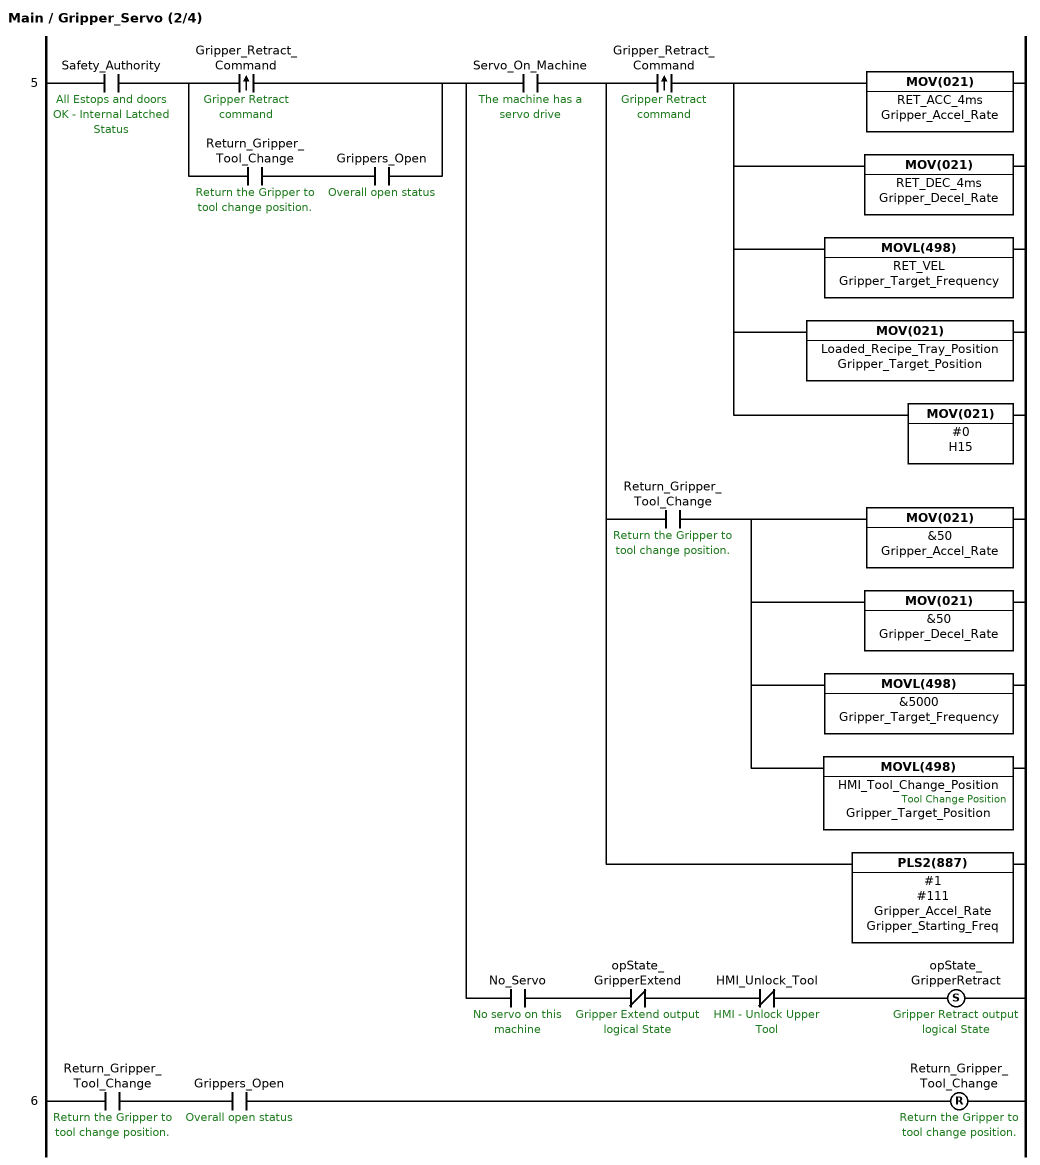
; [picture p96: Main / Gripper_Servo, rungs 5-6]
; rung 5
LD Safety_Authority  ; All Estops and doors OK - Internal Latched Status
@LD Gripper_Retract_Command  ; Gripper Retract command
LD Return_Gripper_Tool_Change  ; Return the Gripper to tool change position.
AND Grippers_Open  ; Overall open status
ORLD
ANDLD
OUT TR0
AND Servo_On_Machine  ; The machine has a servo drive
OUT TR1
@AND Gripper_Retract_Command  ; Gripper Retract command
MOV(021) RET_ACC_4ms Gripper_Accel_Rate
MOV(021) RET_DEC_4ms Gripper_Decel_Rate
MOVL(498) RET_VEL Gripper_Target_Frequency
MOV(021) Loaded_Recipe_Tray_Position Gripper_Target_Position
MOV(021) #0 H15
LD TR1
AND Return_Gripper_Tool_Change  ; Return the Gripper to tool change position.
MOV(021) &50 Gripper_Accel_Rate
MOV(021) &50 Gripper_Decel_Rate
MOVL(498) &5000 Gripper_Target_Frequency
MOVL(498) HMI_Tool_Change_Position Gripper_Target_Position  ; Tool Change Position
LD TR1
PLS2(887) #1 #111 Gripper_Accel_Rate Gripper_Starting_Freq
LD TR0
AND No_Servo  ; No servo on this machine
ANDNOT opState_GripperExtend  ; Gripper Extend output logical State
ANDNOT HMI_Unlock_Tool  ; HMI - Unlock Upper Tool
SET opState_GripperRetract  ; Gripper Retract output logical State
; rung 6
LD Return_Gripper_Tool_Change  ; Return the Gripper to tool change position.
AND Grippers_Open  ; Overall open status
RSET Return_Gripper_Tool_Change  ; Return the Gripper to tool change position.

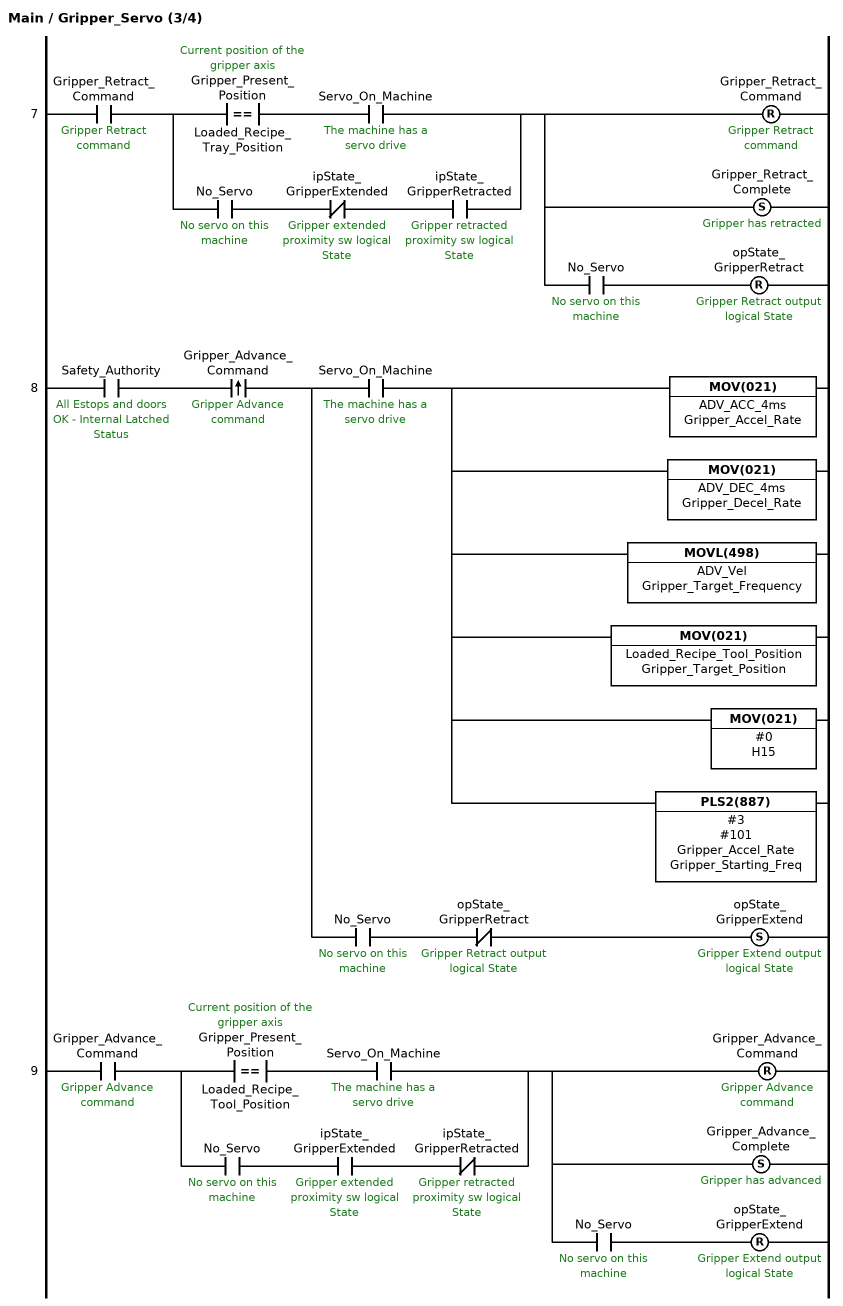
; rung 7
LD Gripper_Retract_Command  ; Gripper Retract command
LD=(300) Gripper_Present_Position Loaded_Recipe_Tray_Position  ; Current position of the gripper axis
AND Servo_On_Machine  ; The machine has a servo drive
LD No_Servo  ; No servo on this machine
ANDNOT ipState_GripperExtended  ; Gripper extended proximity sw logical State
AND ipState_GripperRetracted  ; Gripper retracted proximity sw logical State
ORLD
ANDLD
RSET Gripper_Retract_Command  ; Gripper Retract command
SET Gripper_Retract_Complete  ; Gripper has retracted
AND No_Servo  ; No servo on this machine
RSET opState_GripperRetract  ; Gripper Retract output logical State
; rung 8
LD Safety_Authority  ; All Estops and doors OK - Internal Latched Status
@AND Gripper_Advance_Command  ; Gripper Advance command
OUT TR0
AND Servo_On_Machine  ; The machine has a servo drive
MOV(021) ADV_ACC_4ms Gripper_Accel_Rate
MOV(021) ADV_DEC_4ms Gripper_Decel_Rate
MOVL(498) ADV_Vel Gripper_Target_Frequency
MOV(021) Loaded_Recipe_Tool_Position Gripper_Target_Position
MOV(021) #0 H15
PLS2(887) #3 #101 Gripper_Accel_Rate Gripper_Starting_Freq
LD TR0
AND No_Servo  ; No servo on this machine
ANDNOT opState_GripperRetract  ; Gripper Retract output logical State
SET opState_GripperExtend  ; Gripper Extend output logical State
; rung 9
LD Gripper_Advance_Command  ; Gripper Advance command
LD=(300) Gripper_Present_Position Loaded_Recipe_Tool_Position  ; Current position of the gripper axis
AND Servo_On_Machine  ; The machine has a servo drive
LD No_Servo  ; No servo on this machine
AND ipState_GripperExtended  ; Gripper extended proximity sw logical State
ANDNOT ipState_GripperRetracted  ; Gripper retracted proximity sw logical State
ORLD
ANDLD
RSET Gripper_Advance_Command  ; Gripper Advance command
SET Gripper_Advance_Complete  ; Gripper has advanced
AND No_Servo  ; No servo on this machine
RSET opState_GripperExtend  ; Gripper Extend output logical State

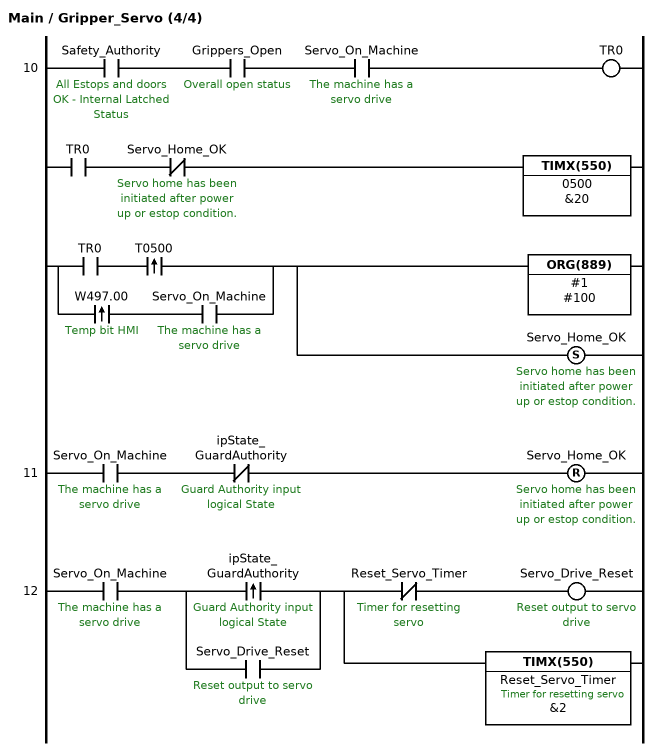
; rung 10
LD Safety_Authority  ; All Estops and doors OK - Internal Latched Status
AND Grippers_Open  ; Overall open status
AND Servo_On_Machine  ; The machine has a servo drive
OUT TR0
ANDNOT Servo_Home_OK  ; Servo home has been initiated after power up or estop condition.
TIMX(550) 0500 &20
LD TR0
@AND T0500
@LD W497.00  ; Temp bit HMI
AND Servo_On_Machine  ; The machine has a servo drive
ORLD
ORG(889) #1 #100
SET Servo_Home_OK  ; Servo home has been initiated after power up or estop condition.
; rung 11
LD Servo_On_Machine  ; The machine has a servo drive
ANDNOT ipState_GuardAuthority  ; Guard Authority input logical State
RSET Servo_Home_OK  ; Servo home has been initiated after power up or estop condition.
; rung 12
LD Servo_On_Machine  ; The machine has a servo drive
@LD ipState_GuardAuthority  ; Guard Authority input logical State
OR Servo_Drive_Reset  ; Reset output to servo drive
ANDLD
OUT TR0
ANDNOT Reset_Servo_Timer  ; Timer for resetting servo
OUT Servo_Drive_Reset  ; Reset output to servo drive
LD TR0
TIMX(550) Reset_Servo_Timer &2  ; Timer for resetting servo

### Section Temp_Control_and_Analog

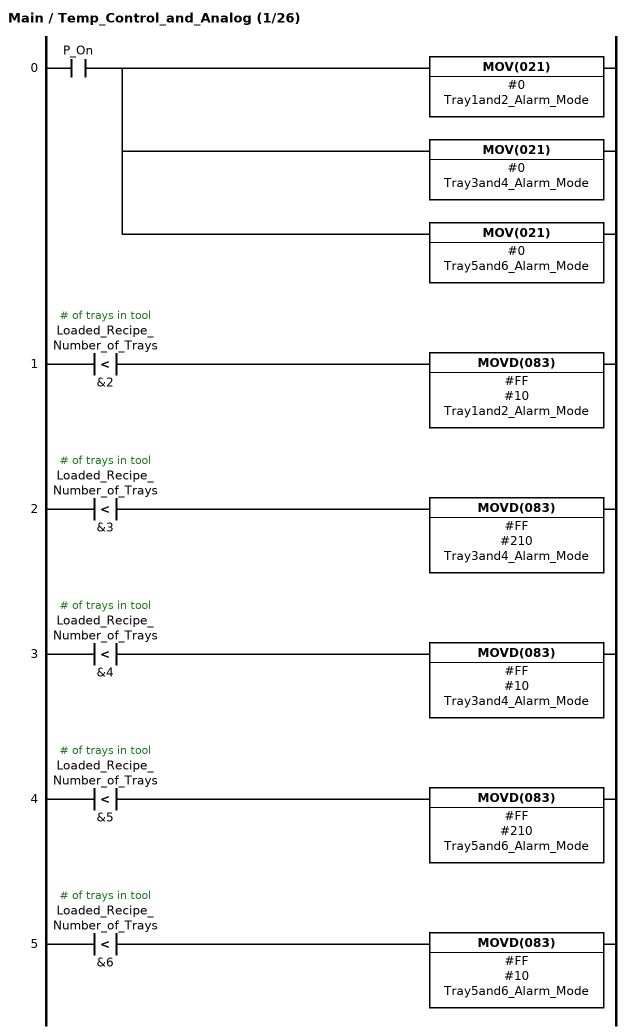
; rung 0
LD P_On
MOV(021) #0 Tray1and2_Alarm_Mode
MOV(021) #0 Tray3and4_Alarm_Mode
MOV(021) #0 Tray5and6_Alarm_Mode
; rung 1
LD<(310) Loaded_Recipe_Number_of_Trays &2  ; # of trays in tool
MOVD(083) #FF #10 Tray1and2_Alarm_Mode
; rung 2
LD<(310) Loaded_Recipe_Number_of_Trays &3  ; # of trays in tool
MOVD(083) #FF #210 Tray3and4_Alarm_Mode
; rung 3
LD<(310) Loaded_Recipe_Number_of_Trays &4  ; # of trays in tool
MOVD(083) #FF #10 Tray3and4_Alarm_Mode
; rung 4
LD<(310) Loaded_Recipe_Number_of_Trays &5  ; # of trays in tool
MOVD(083) #FF #210 Tray5and6_Alarm_Mode
; rung 5
LD<(310) Loaded_Recipe_Number_of_Trays &6  ; # of trays in tool
MOVD(083) #FF #10 Tray5and6_Alarm_Mode

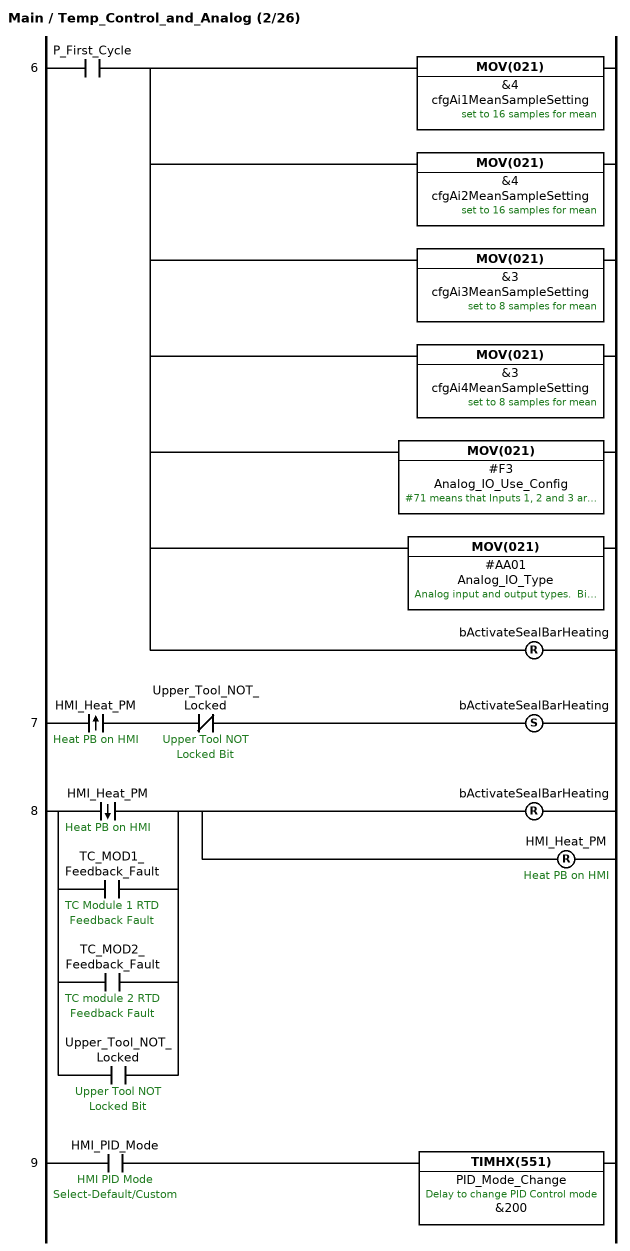
; rung 6
LD P_First_Cycle
MOV(021) &4 cfgAi1MeanSampleSetting  ; set to 16 samples for mean
MOV(021) &4 cfgAi2MeanSampleSetting  ; set to 16 samples for mean
MOV(021) &3 cfgAi3MeanSampleSetting  ; set to 8 samples for mean
MOV(021) &3 cfgAi4MeanSampleSetting  ; set to 8 samples for mean
MOV(021) #F3 Analog_IO_Use_Config  ; #71 means that Inputs 1, 2 and 3 are used (bits 4, 5 and 6 on makes up 7 HEX) and output 1 is used (bit 0 on makes up 1 HEX).
MOV(021) #AA01 Analog_IO_Type  ; Analog input and output types.  Bit pattern of 1010101000000001 (#AA01) means all inputs are 4-20 mA and the output are 0 - 10VDC).
RSET bActivateSealBarHeating
; rung 7
@LD HMI_Heat_PM  ; Heat PB on HMI
ANDNOT Upper_Tool_NOT_Locked  ; Upper Tool NOT Locked Bit
SET bActivateSealBarHeating
; rung 8
%LD HMI_Heat_PM  ; Heat PB on HMI
OR TC_MOD1_Feedback_Fault  ; TC Module 1 RTD Feedback Fault
OR TC_MOD2_Feedback_Fault  ; TC module 2 RTD Feedback Fault
OR Upper_Tool_NOT_Locked  ; Upper Tool NOT Locked Bit
RSET bActivateSealBarHeating
RSET HMI_Heat_PM  ; Heat PB on HMI
; rung 9
LD HMI_PID_Mode  ; HMI PID Mode Select-Default/Custom
TIMHX(551) PID_Mode_Change &200  ; Delay to change PID Control mode

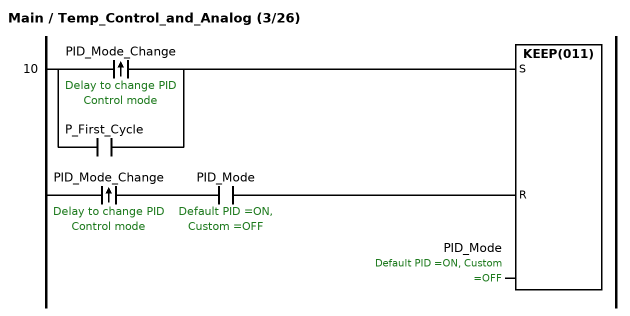
; rung 10
@LD PID_Mode_Change  ; Delay to change PID Control mode
OR P_First_Cycle
@LD PID_Mode_Change  ; Delay to change PID Control mode
AND PID_Mode  ; Default PID =ON, Custom =OFF
KEEP(011) PID_Mode  ; Default PID =ON, Custom =OFF

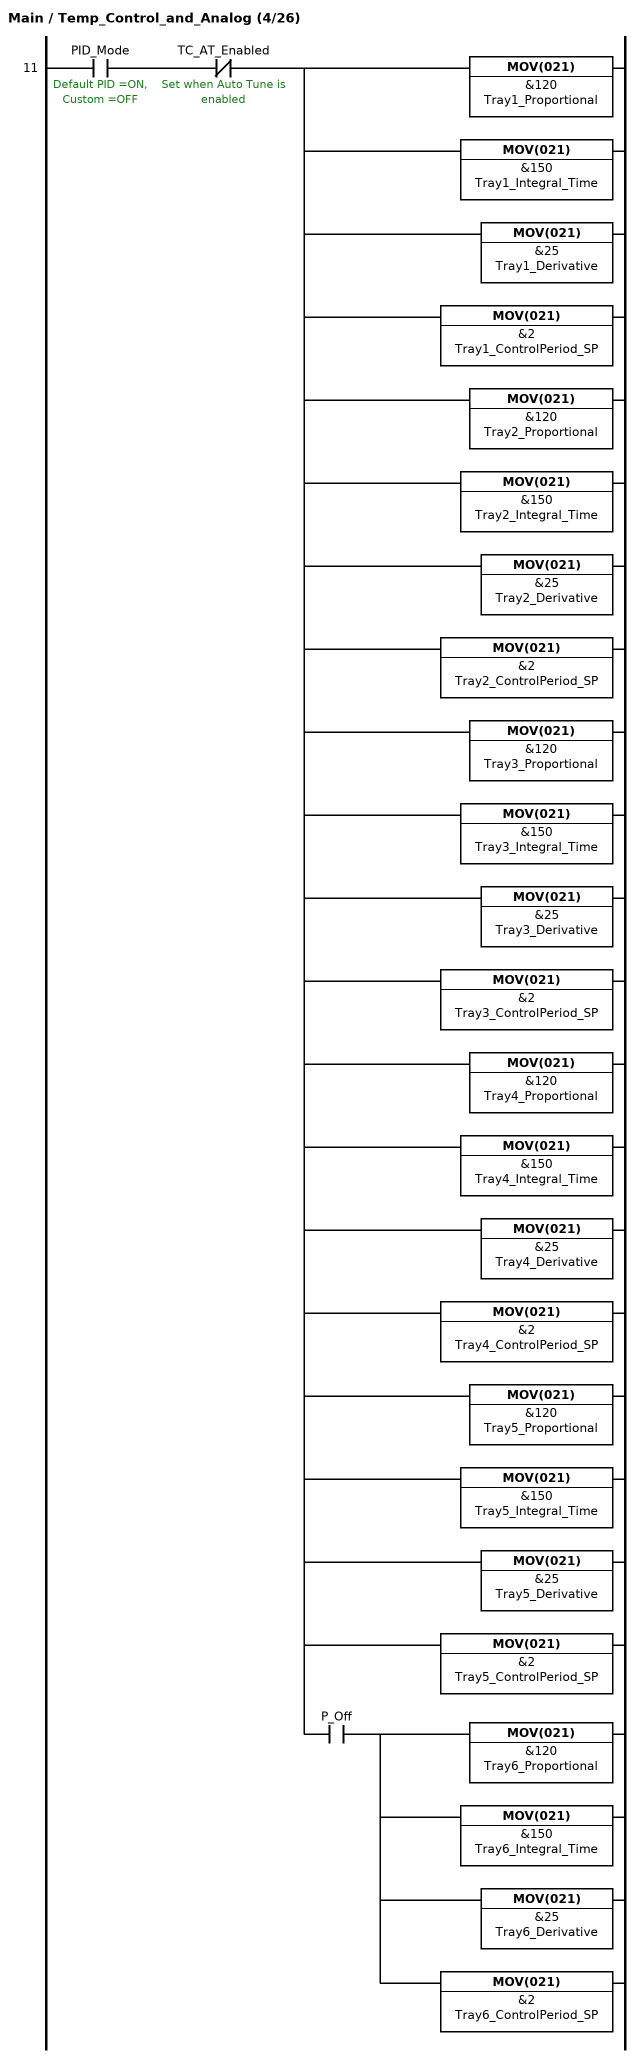
; rung 11
LD PID_Mode  ; Default PID =ON, Custom =OFF
ANDNOT TC_AT_Enabled  ; Set when Auto Tune is enabled
MOV(021) &120 Tray1_Proportional
MOV(021) &150 Tray1_Integral_Time
MOV(021) &25 Tray1_Derivative
MOV(021) &2 Tray1_ControlPeriod_SP
MOV(021) &120 Tray2_Proportional
MOV(021) &150 Tray2_Integral_Time
MOV(021) &25 Tray2_Derivative
MOV(021) &2 Tray2_ControlPeriod_SP
MOV(021) &120 Tray3_Proportional
MOV(021) &150 Tray3_Integral_Time
MOV(021) &25 Tray3_Derivative
MOV(021) &2 Tray3_ControlPeriod_SP
MOV(021) &120 Tray4_Proportional
MOV(021) &150 Tray4_Integral_Time
MOV(021) &25 Tray4_Derivative
MOV(021) &2 Tray4_ControlPeriod_SP
MOV(021) &120 Tray5_Proportional
MOV(021) &150 Tray5_Integral_Time
MOV(021) &25 Tray5_Derivative
MOV(021) &2 Tray5_ControlPeriod_SP
AND P_Off
MOV(021) &120 Tray6_Proportional
MOV(021) &150 Tray6_Integral_Time
MOV(021) &25 Tray6_Derivative
MOV(021) &2 Tray6_ControlPeriod_SP

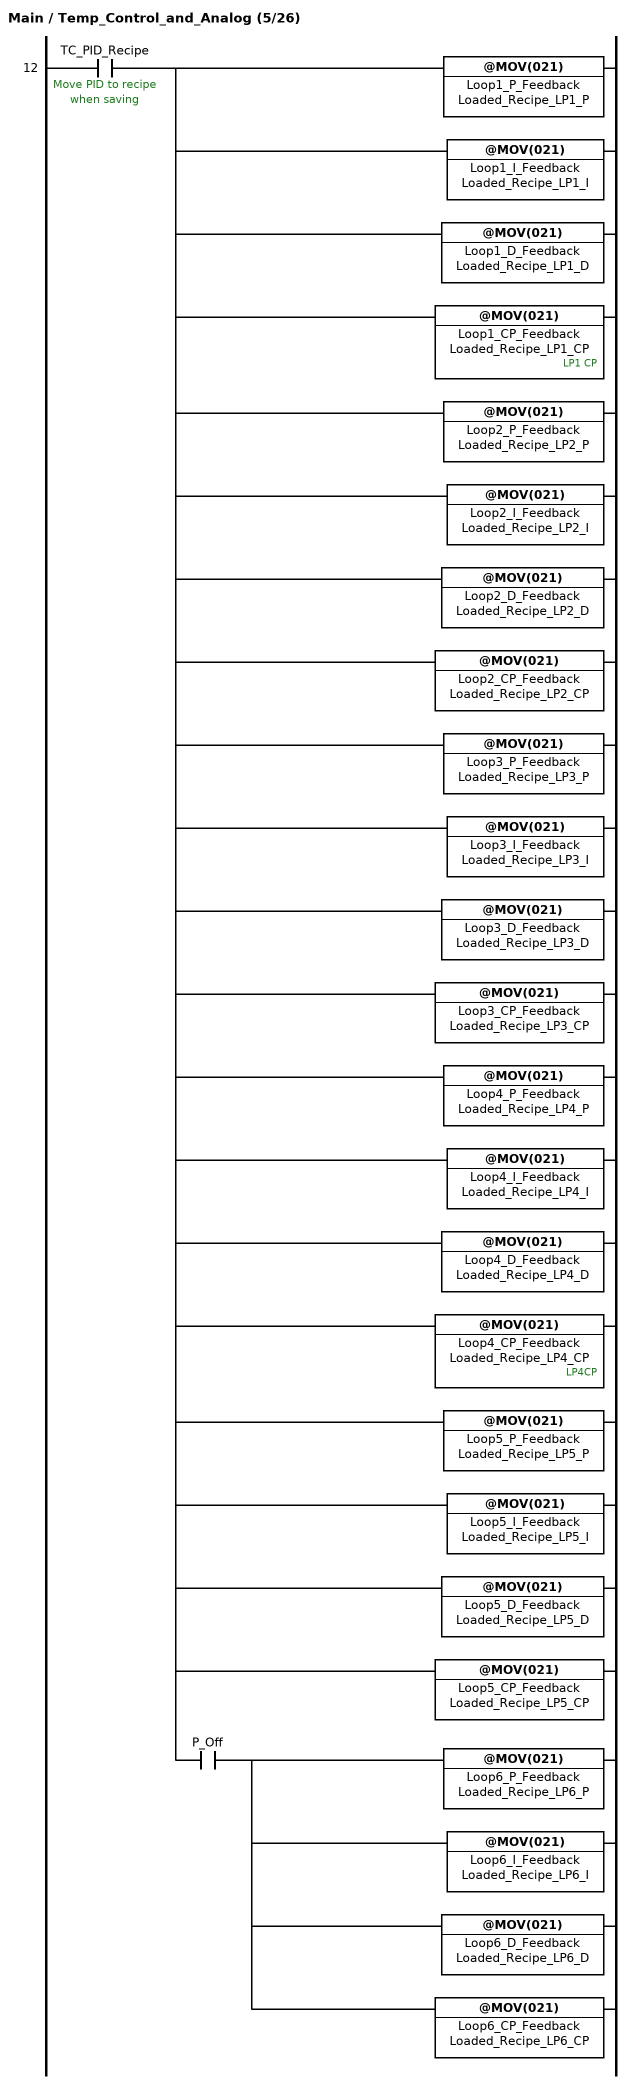
; rung 12
LD TC_PID_Recipe  ; Move PID to recipe when saving
@MOV(021) Loop1_P_Feedback Loaded_Recipe_LP1_P
@MOV(021) Loop1_I_Feedback Loaded_Recipe_LP1_I
@MOV(021) Loop1_D_Feedback Loaded_Recipe_LP1_D
@MOV(021) Loop1_CP_Feedback Loaded_Recipe_LP1_CP  ; LP1 CP
@MOV(021) Loop2_P_Feedback Loaded_Recipe_LP2_P
@MOV(021) Loop2_I_Feedback Loaded_Recipe_LP2_I
@MOV(021) Loop2_D_Feedback Loaded_Recipe_LP2_D
@MOV(021) Loop2_CP_Feedback Loaded_Recipe_LP2_CP
@MOV(021) Loop3_P_Feedback Loaded_Recipe_LP3_P
@MOV(021) Loop3_I_Feedback Loaded_Recipe_LP3_I
@MOV(021) Loop3_D_Feedback Loaded_Recipe_LP3_D
@MOV(021) Loop3_CP_Feedback Loaded_Recipe_LP3_CP
@MOV(021) Loop4_P_Feedback Loaded_Recipe_LP4_P
@MOV(021) Loop4_I_Feedback Loaded_Recipe_LP4_I
@MOV(021) Loop4_D_Feedback Loaded_Recipe_LP4_D
@MOV(021) Loop4_CP_Feedback Loaded_Recipe_LP4_CP  ; LP4CP
@MOV(021) Loop5_P_Feedback Loaded_Recipe_LP5_P
@MOV(021) Loop5_I_Feedback Loaded_Recipe_LP5_I
@MOV(021) Loop5_D_Feedback Loaded_Recipe_LP5_D
@MOV(021) Loop5_CP_Feedback Loaded_Recipe_LP5_CP
AND P_Off
@MOV(021) Loop6_P_Feedback Loaded_Recipe_LP6_P
@MOV(021) Loop6_I_Feedback Loaded_Recipe_LP6_I
@MOV(021) Loop6_D_Feedback Loaded_Recipe_LP6_D
@MOV(021) Loop6_CP_Feedback Loaded_Recipe_LP6_CP

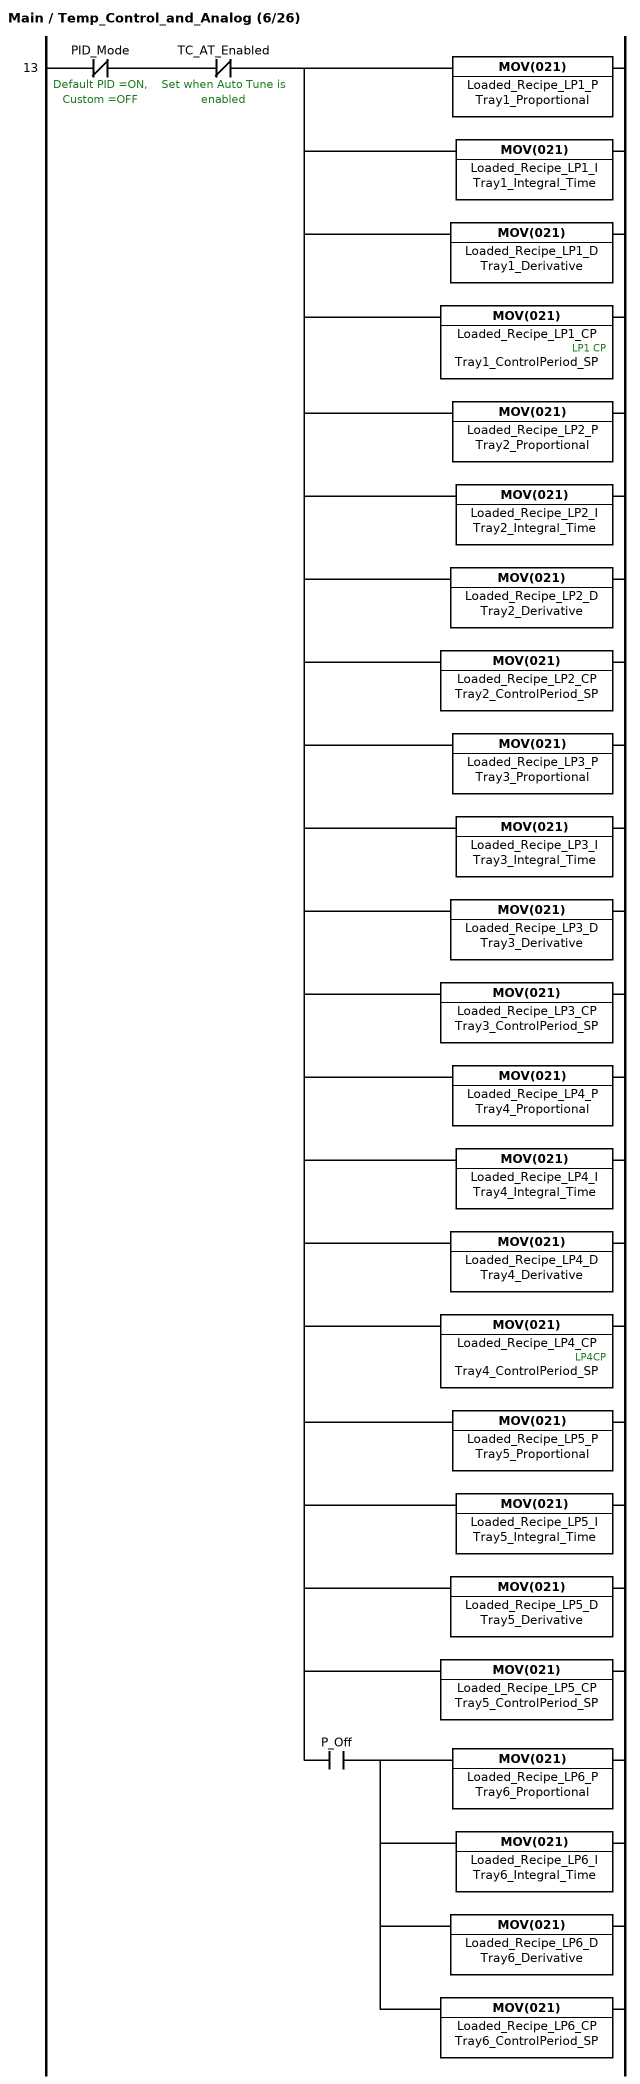
; rung 13
LDNOT PID_Mode  ; Default PID =ON, Custom =OFF
ANDNOT TC_AT_Enabled  ; Set when Auto Tune is enabled
MOV(021) Loaded_Recipe_LP1_P Tray1_Proportional
MOV(021) Loaded_Recipe_LP1_I Tray1_Integral_Time
MOV(021) Loaded_Recipe_LP1_D Tray1_Derivative
MOV(021) Loaded_Recipe_LP1_CP Tray1_ControlPeriod_SP  ; LP1 CP
MOV(021) Loaded_Recipe_LP2_P Tray2_Proportional
MOV(021) Loaded_Recipe_LP2_I Tray2_Integral_Time
MOV(021) Loaded_Recipe_LP2_D Tray2_Derivative
MOV(021) Loaded_Recipe_LP2_CP Tray2_ControlPeriod_SP
MOV(021) Loaded_Recipe_LP3_P Tray3_Proportional
MOV(021) Loaded_Recipe_LP3_I Tray3_Integral_Time
MOV(021) Loaded_Recipe_LP3_D Tray3_Derivative
MOV(021) Loaded_Recipe_LP3_CP Tray3_ControlPeriod_SP
MOV(021) Loaded_Recipe_LP4_P Tray4_Proportional
MOV(021) Loaded_Recipe_LP4_I Tray4_Integral_Time
MOV(021) Loaded_Recipe_LP4_D Tray4_Derivative
MOV(021) Loaded_Recipe_LP4_CP Tray4_ControlPeriod_SP  ; LP4CP
MOV(021) Loaded_Recipe_LP5_P Tray5_Proportional
MOV(021) Loaded_Recipe_LP5_I Tray5_Integral_Time
MOV(021) Loaded_Recipe_LP5_D Tray5_Derivative
MOV(021) Loaded_Recipe_LP5_CP Tray5_ControlPeriod_SP
AND P_Off
MOV(021) Loaded_Recipe_LP6_P Tray6_Proportional
MOV(021) Loaded_Recipe_LP6_I Tray6_Integral_Time
MOV(021) Loaded_Recipe_LP6_D Tray6_Derivative
MOV(021) Loaded_Recipe_LP6_CP Tray6_ControlPeriod_SP

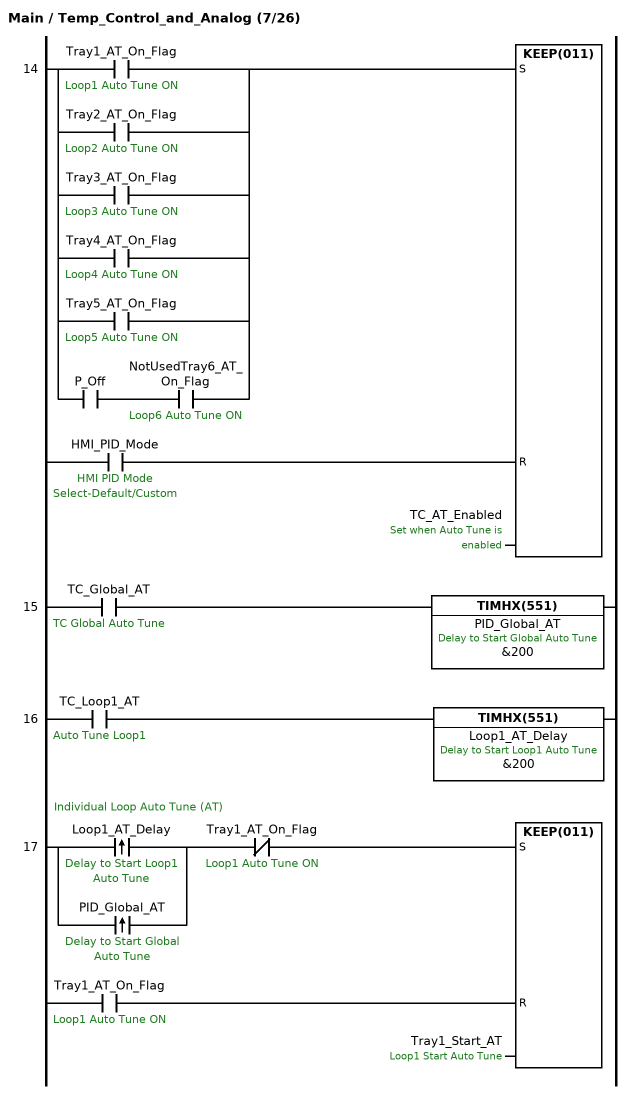
; rung 14
LD Tray1_AT_On_Flag  ; Loop1 Auto Tune ON
OR Tray2_AT_On_Flag  ; Loop2 Auto Tune ON
OR Tray3_AT_On_Flag  ; Loop3 Auto Tune ON
OR Tray4_AT_On_Flag  ; Loop4 Auto Tune ON
OR Tray5_AT_On_Flag  ; Loop5 Auto Tune ON
LD P_Off
AND NotUsedTray6_AT_On_Flag  ; Loop6 Auto Tune ON
ORLD
LD HMI_PID_Mode  ; HMI PID Mode Select-Default/Custom
KEEP(011) TC_AT_Enabled  ; Set when Auto Tune is enabled
; rung 15
LD TC_Global_AT  ; TC Global Auto Tune
TIMHX(551) PID_Global_AT &200  ; Delay to Start Global Auto Tune
; rung 16
LD TC_Loop1_AT  ; Auto Tune Loop1
TIMHX(551) Loop1_AT_Delay &200  ; Delay to Start Loop1 Auto Tune
; rung 17: Individual Loop Auto Tune (AT)
@LD Loop1_AT_Delay  ; Delay to Start Loop1 Auto Tune
@OR PID_Global_AT  ; Delay to Start Global Auto Tune
ANDNOT Tray1_AT_On_Flag  ; Loop1 Auto Tune ON
LD Tray1_AT_On_Flag  ; Loop1 Auto Tune ON
KEEP(011) Tray1_Start_AT  ; Loop1 Start Auto Tune

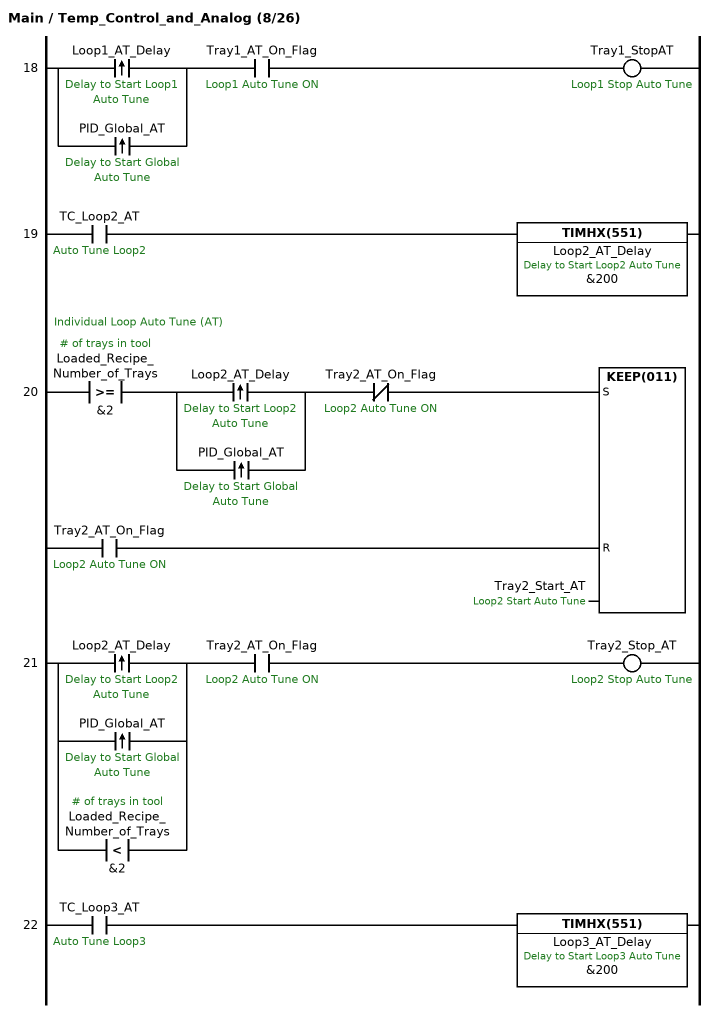
; rung 18
@LD Loop1_AT_Delay  ; Delay to Start Loop1 Auto Tune
@OR PID_Global_AT  ; Delay to Start Global Auto Tune
AND Tray1_AT_On_Flag  ; Loop1 Auto Tune ON
OUT Tray1_StopAT  ; Loop1 Stop Auto Tune
; rung 19
LD TC_Loop2_AT  ; Auto Tune Loop2
TIMHX(551) Loop2_AT_Delay &200  ; Delay to Start Loop2 Auto Tune
; rung 20: Individual Loop Auto Tune (AT)
LD>=(325) Loaded_Recipe_Number_of_Trays &2  ; # of trays in tool
@LD Loop2_AT_Delay  ; Delay to Start Loop2 Auto Tune
@OR PID_Global_AT  ; Delay to Start Global Auto Tune
ANDLD
ANDNOT Tray2_AT_On_Flag  ; Loop2 Auto Tune ON
LD Tray2_AT_On_Flag  ; Loop2 Auto Tune ON
KEEP(011) Tray2_Start_AT  ; Loop2 Start Auto Tune
; rung 21
@LD Loop2_AT_Delay  ; Delay to Start Loop2 Auto Tune
@OR PID_Global_AT  ; Delay to Start Global Auto Tune
OR<(310) Loaded_Recipe_Number_of_Trays &2  ; # of trays in tool
AND Tray2_AT_On_Flag  ; Loop2 Auto Tune ON
OUT Tray2_Stop_AT  ; Loop2 Stop Auto Tune
; rung 22
LD TC_Loop3_AT  ; Auto Tune Loop3
TIMHX(551) Loop3_AT_Delay &200  ; Delay to Start Loop3 Auto Tune

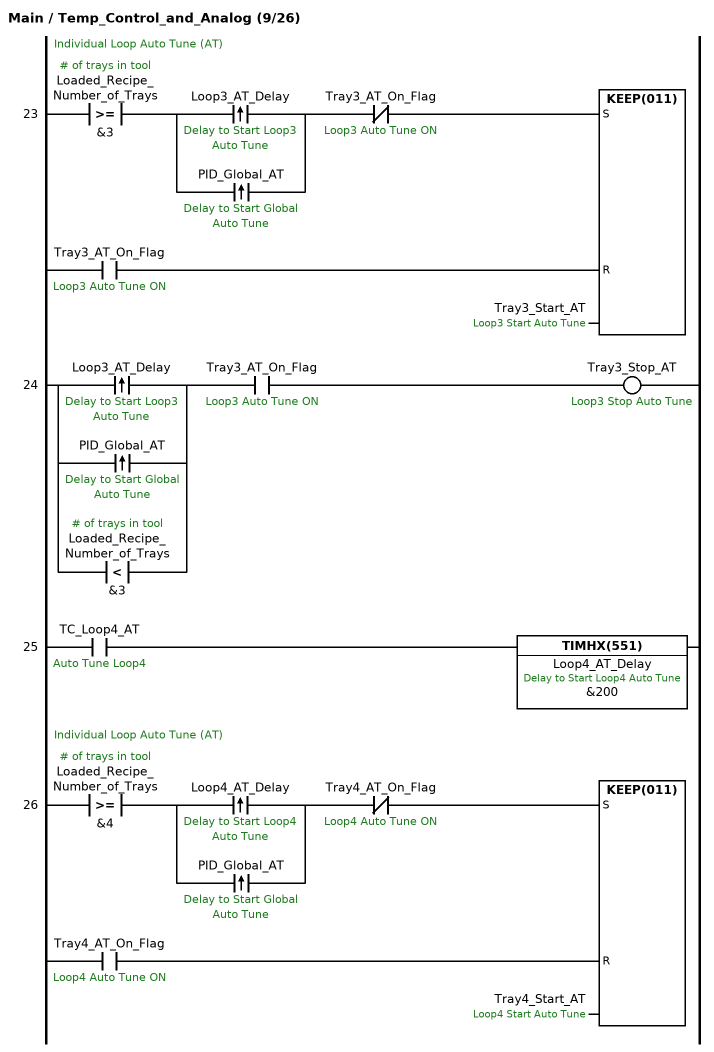
; rung 23: Individual Loop Auto Tune (AT)
LD>=(325) Loaded_Recipe_Number_of_Trays &3  ; # of trays in tool
@LD Loop3_AT_Delay  ; Delay to Start Loop3 Auto Tune
@OR PID_Global_AT  ; Delay to Start Global Auto Tune
ANDLD
ANDNOT Tray3_AT_On_Flag  ; Loop3 Auto Tune ON
LD Tray3_AT_On_Flag  ; Loop3 Auto Tune ON
KEEP(011) Tray3_Start_AT  ; Loop3 Start Auto Tune
; rung 24
@LD Loop3_AT_Delay  ; Delay to Start Loop3 Auto Tune
@OR PID_Global_AT  ; Delay to Start Global Auto Tune
OR<(310) Loaded_Recipe_Number_of_Trays &3  ; # of trays in tool
AND Tray3_AT_On_Flag  ; Loop3 Auto Tune ON
OUT Tray3_Stop_AT  ; Loop3 Stop Auto Tune
; rung 25
LD TC_Loop4_AT  ; Auto Tune Loop4
TIMHX(551) Loop4_AT_Delay &200  ; Delay to Start Loop4 Auto Tune
; rung 26: Individual Loop Auto Tune (AT)
LD>=(325) Loaded_Recipe_Number_of_Trays &4  ; # of trays in tool
@LD Loop4_AT_Delay  ; Delay to Start Loop4 Auto Tune
@OR PID_Global_AT  ; Delay to Start Global Auto Tune
ANDLD
ANDNOT Tray4_AT_On_Flag  ; Loop4 Auto Tune ON
LD Tray4_AT_On_Flag  ; Loop4 Auto Tune ON
KEEP(011) Tray4_Start_AT  ; Loop4 Start Auto Tune

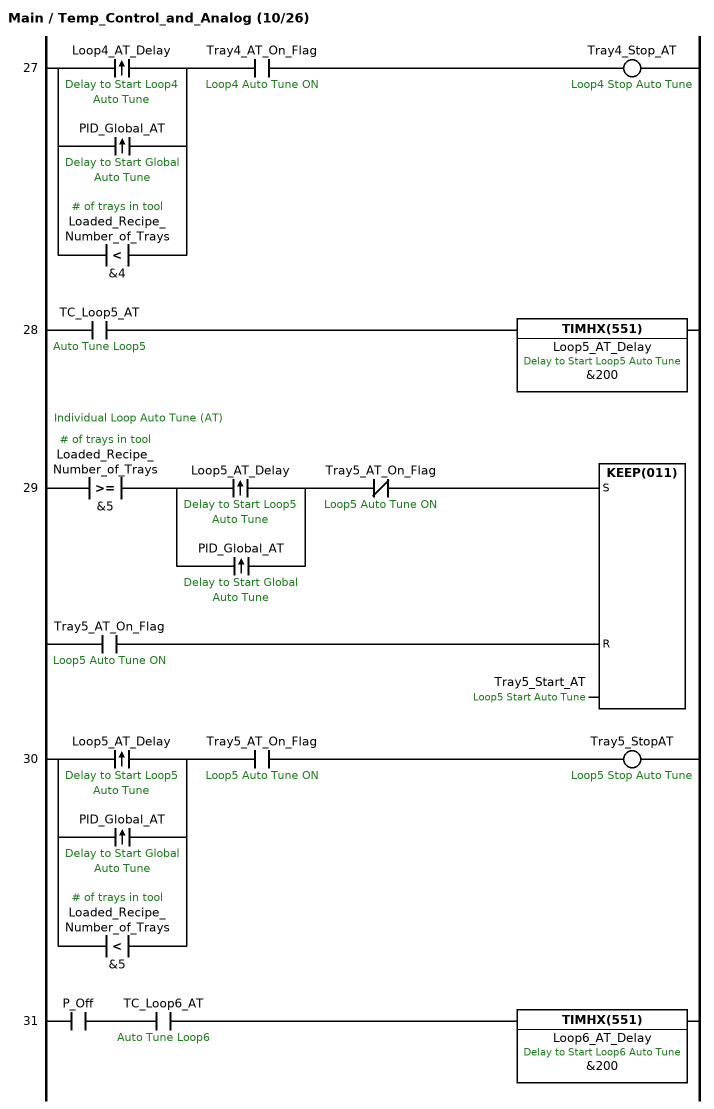
; rung 27
@LD Loop4_AT_Delay  ; Delay to Start Loop4 Auto Tune
@OR PID_Global_AT  ; Delay to Start Global Auto Tune
OR<(310) Loaded_Recipe_Number_of_Trays &4  ; # of trays in tool
AND Tray4_AT_On_Flag  ; Loop4 Auto Tune ON
OUT Tray4_Stop_AT  ; Loop4 Stop Auto Tune
; rung 28
LD TC_Loop5_AT  ; Auto Tune Loop5
TIMHX(551) Loop5_AT_Delay &200  ; Delay to Start Loop5 Auto Tune
; rung 29: Individual Loop Auto Tune (AT)
LD>=(325) Loaded_Recipe_Number_of_Trays &5  ; # of trays in tool
@LD Loop5_AT_Delay  ; Delay to Start Loop5 Auto Tune
@OR PID_Global_AT  ; Delay to Start Global Auto Tune
ANDLD
ANDNOT Tray5_AT_On_Flag  ; Loop5 Auto Tune ON
LD Tray5_AT_On_Flag  ; Loop5 Auto Tune ON
KEEP(011) Tray5_Start_AT  ; Loop5 Start Auto Tune
; rung 30
@LD Loop5_AT_Delay  ; Delay to Start Loop5 Auto Tune
@OR PID_Global_AT  ; Delay to Start Global Auto Tune
OR<(310) Loaded_Recipe_Number_of_Trays &5  ; # of trays in tool
AND Tray5_AT_On_Flag  ; Loop5 Auto Tune ON
OUT Tray5_StopAT  ; Loop5 Stop Auto Tune
; rung 31
LD P_Off
AND TC_Loop6_AT  ; Auto Tune Loop6
TIMHX(551) Loop6_AT_Delay &200  ; Delay to Start Loop6 Auto Tune

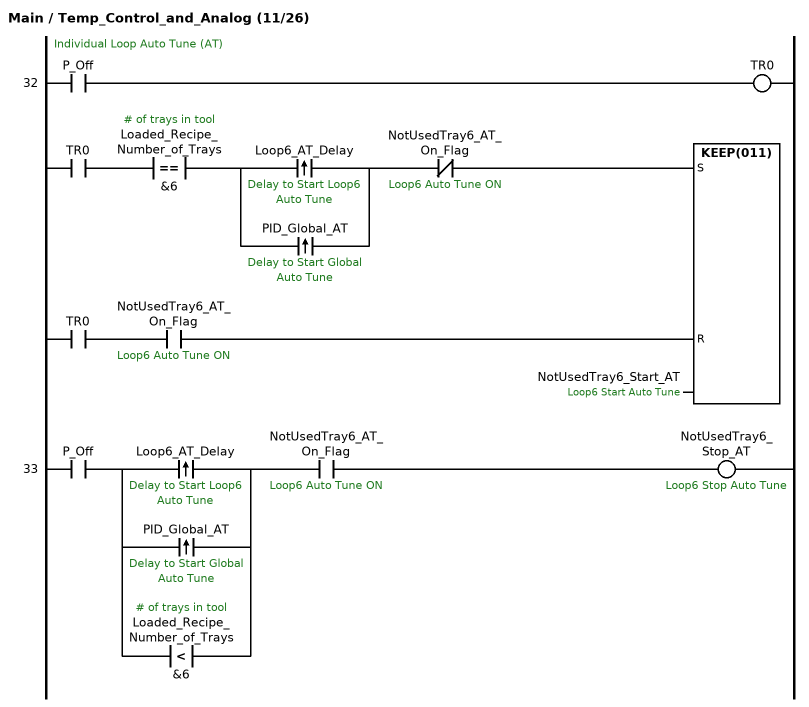
; rung 32: Individual Loop Auto Tune (AT)
LD P_Off
OUT TR0
AND=(300) Loaded_Recipe_Number_of_Trays &6  ; # of trays in tool
@LD Loop6_AT_Delay  ; Delay to Start Loop6 Auto Tune
@OR PID_Global_AT  ; Delay to Start Global Auto Tune
ANDLD
ANDNOT NotUsedTray6_AT_On_Flag  ; Loop6 Auto Tune ON
LD TR0
AND NotUsedTray6_AT_On_Flag  ; Loop6 Auto Tune ON
KEEP(011) NotUsedTray6_Start_AT  ; Loop6 Start Auto Tune
; rung 33
LD P_Off
@LD Loop6_AT_Delay  ; Delay to Start Loop6 Auto Tune
@OR PID_Global_AT  ; Delay to Start Global Auto Tune
OR<(310) Loaded_Recipe_Number_of_Trays &6  ; # of trays in tool
ANDLD
AND NotUsedTray6_AT_On_Flag  ; Loop6 Auto Tune ON
OUT NotUsedTray6_Stop_AT  ; Loop6 Stop Auto Tune

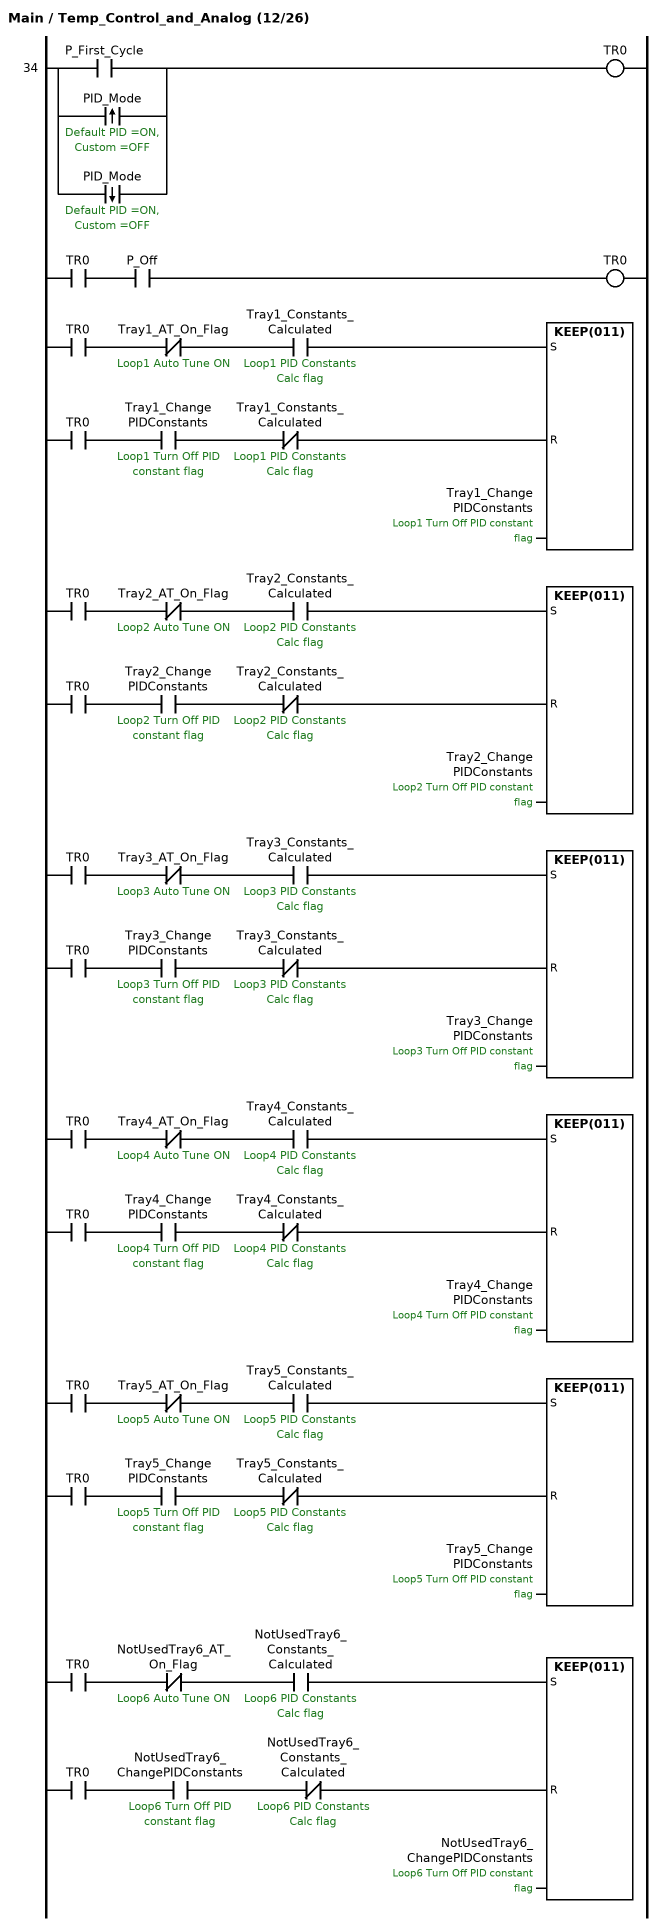
; rung 34
LD P_First_Cycle
@OR PID_Mode  ; Default PID =ON, Custom =OFF
%OR PID_Mode  ; Default PID =ON, Custom =OFF
OUT TR0
ANDNOT Tray1_AT_On_Flag  ; Loop1 Auto Tune ON
AND Tray1_Constants_Calculated  ; Loop1 PID Constants Calc flag
LD TR0
AND Tray1_ChangePIDConstants  ; Loop1 Turn Off PID constant flag
ANDNOT Tray1_Constants_Calculated  ; Loop1 PID Constants Calc flag
KEEP(011) Tray1_ChangePIDConstants  ; Loop1 Turn Off PID constant flag
LD TR0
ANDNOT Tray2_AT_On_Flag  ; Loop2 Auto Tune ON
AND Tray2_Constants_Calculated  ; Loop2 PID Constants Calc flag
LD TR0
AND Tray2_ChangePIDConstants  ; Loop2 Turn Off PID constant flag
ANDNOT Tray2_Constants_Calculated  ; Loop2 PID Constants Calc flag
KEEP(011) Tray2_ChangePIDConstants  ; Loop2 Turn Off PID constant flag
LD TR0
ANDNOT Tray3_AT_On_Flag  ; Loop3 Auto Tune ON
AND Tray3_Constants_Calculated  ; Loop3 PID Constants Calc flag
LD TR0
AND Tray3_ChangePIDConstants  ; Loop3 Turn Off PID constant flag
ANDNOT Tray3_Constants_Calculated  ; Loop3 PID Constants Calc flag
KEEP(011) Tray3_ChangePIDConstants  ; Loop3 Turn Off PID constant flag
LD TR0
ANDNOT Tray4_AT_On_Flag  ; Loop4 Auto Tune ON
AND Tray4_Constants_Calculated  ; Loop4 PID Constants Calc flag
LD TR0
AND Tray4_ChangePIDConstants  ; Loop4 Turn Off PID constant flag
ANDNOT Tray4_Constants_Calculated  ; Loop4 PID Constants Calc flag
KEEP(011) Tray4_ChangePIDConstants  ; Loop4 Turn Off PID constant flag
LD TR0
ANDNOT Tray5_AT_On_Flag  ; Loop5 Auto Tune ON
AND Tray5_Constants_Calculated  ; Loop5 PID Constants Calc flag
LD TR0
AND Tray5_ChangePIDConstants  ; Loop5 Turn Off PID constant flag
ANDNOT Tray5_Constants_Calculated  ; Loop5 PID Constants Calc flag
KEEP(011) Tray5_ChangePIDConstants  ; Loop5 Turn Off PID constant flag
LD TR0
AND P_Off
OUT TR0
ANDNOT NotUsedTray6_AT_On_Flag  ; Loop6 Auto Tune ON
AND NotUsedTray6_Constants_Calculated  ; Loop6 PID Constants Calc flag
LD TR0
AND NotUsedTray6_ChangePIDConstants  ; Loop6 Turn Off PID constant flag
ANDNOT NotUsedTray6_Constants_Calculated  ; Loop6 PID Constants Calc flag
KEEP(011) NotUsedTray6_ChangePIDConstants  ; Loop6 Turn Off PID constant flag

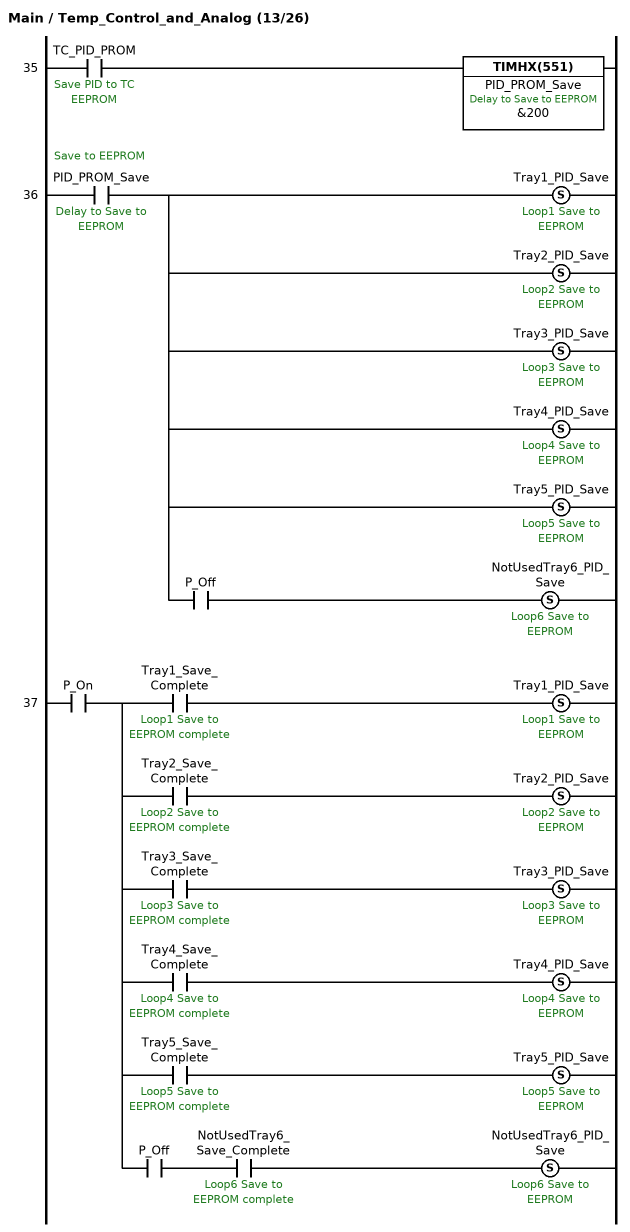
; rung 35
LD TC_PID_PROM  ; Save PID to TC EEPROM
TIMHX(551) PID_PROM_Save &200  ; Delay to Save to EEPROM
; rung 36: Save to EEPROM
LD PID_PROM_Save  ; Delay to Save to EEPROM
SET Tray1_PID_Save  ; Loop1 Save to EEPROM
SET Tray2_PID_Save  ; Loop2 Save to EEPROM
SET Tray3_PID_Save  ; Loop3 Save to EEPROM
SET Tray4_PID_Save  ; Loop4 Save to EEPROM
SET Tray5_PID_Save  ; Loop5 Save to EEPROM
AND P_Off
SET NotUsedTray6_PID_Save  ; Loop6 Save to EEPROM
; rung 37
LD P_On
OUT TR0
AND Tray1_Save_Complete  ; Loop1 Save to EEPROM complete
SET Tray1_PID_Save  ; Loop1 Save to EEPROM
LD TR0
AND Tray2_Save_Complete  ; Loop2 Save to EEPROM complete
SET Tray2_PID_Save  ; Loop2 Save to EEPROM
LD TR0
AND Tray3_Save_Complete  ; Loop3 Save to EEPROM complete
SET Tray3_PID_Save  ; Loop3 Save to EEPROM
LD TR0
AND Tray4_Save_Complete  ; Loop4 Save to EEPROM complete
SET Tray4_PID_Save  ; Loop4 Save to EEPROM
LD TR0
AND Tray5_Save_Complete  ; Loop5 Save to EEPROM complete
SET Tray5_PID_Save  ; Loop5 Save to EEPROM
LD TR0
AND P_Off
AND NotUsedTray6_Save_Complete  ; Loop6 Save to EEPROM complete
SET NotUsedTray6_PID_Save  ; Loop6 Save to EEPROM

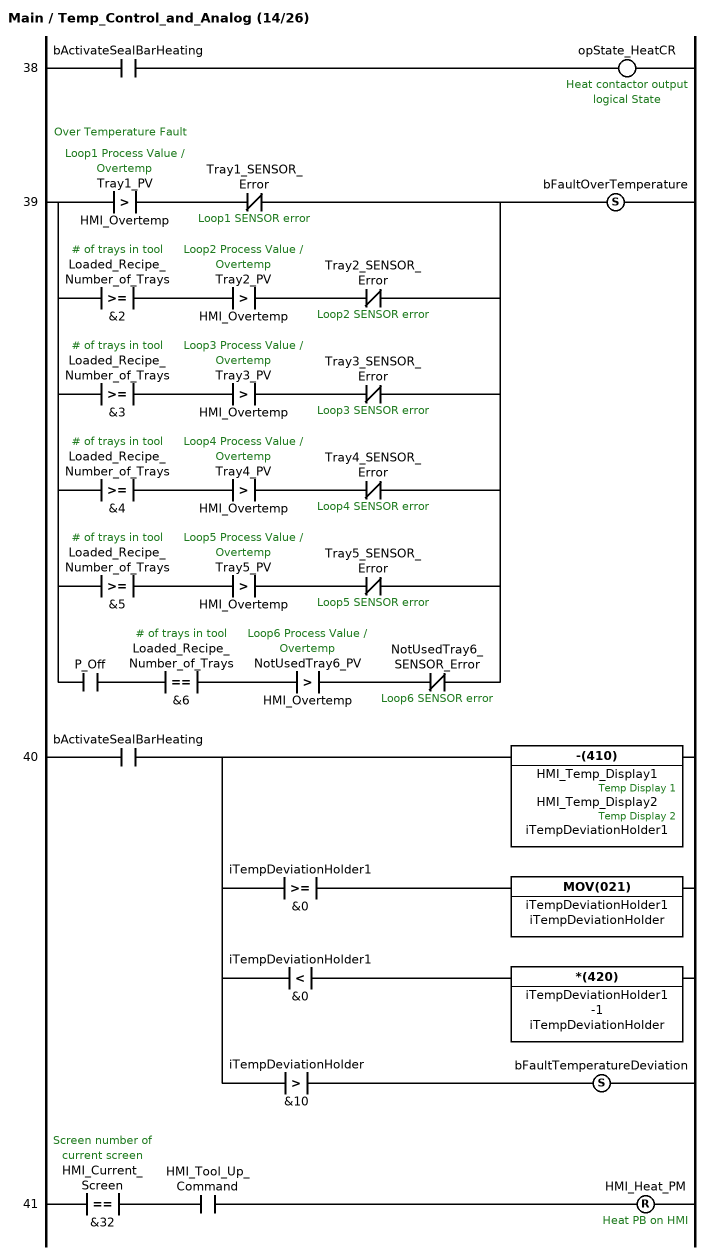
; rung 38
LD bActivateSealBarHeating
OUT opState_HeatCR  ; Heat contactor output logical State
; rung 39: Over Temperature Fault
LD>S(322) Tray1_PV HMI_Overtemp  ; Loop1 Process Value, Overtemp
ANDNOT Tray1_SENSOR_Error  ; Loop1 SENSOR error
LD>=(325) Loaded_Recipe_Number_of_Trays &2  ; # of trays in tool
AND>S(322) Tray2_PV HMI_Overtemp  ; Loop2 Process Value, Overtemp
ANDNOT Tray2_SENSOR_Error  ; Loop2 SENSOR error
ORLD
LD>=(325) Loaded_Recipe_Number_of_Trays &3  ; # of trays in tool
AND>S(322) Tray3_PV HMI_Overtemp  ; Loop3 Process Value, Overtemp
ANDNOT Tray3_SENSOR_Error  ; Loop3 SENSOR error
ORLD
LD>=(325) Loaded_Recipe_Number_of_Trays &4  ; # of trays in tool
AND>S(322) Tray4_PV HMI_Overtemp  ; Loop4 Process Value, Overtemp
ANDNOT Tray4_SENSOR_Error  ; Loop4 SENSOR error
ORLD
LD>=(325) Loaded_Recipe_Number_of_Trays &5  ; # of trays in tool
AND>S(322) Tray5_PV HMI_Overtemp  ; Loop5 Process Value, Overtemp
ANDNOT Tray5_SENSOR_Error  ; Loop5 SENSOR error
ORLD
LD P_Off
AND=(300) Loaded_Recipe_Number_of_Trays &6  ; # of trays in tool
AND>S(322) NotUsedTray6_PV HMI_Overtemp  ; Loop6 Process Value, Overtemp
ANDNOT NotUsedTray6_SENSOR_Error  ; Loop6 SENSOR error
ORLD
SET bFaultOverTemperature
; rung 40
LD bActivateSealBarHeating
OUT TR0
-(410) HMI_Temp_Display1 HMI_Temp_Display2 iTempDeviationHolder1  ; Temp Display 1, Temp Display 2
AND>=(325) iTempDeviationHolder1 &0
MOV(021) iTempDeviationHolder1 iTempDeviationHolder
LD TR0
AND<(310) iTempDeviationHolder1 &0
*(420) iTempDeviationHolder1 -1 iTempDeviationHolder
LD TR0
AND>(320) iTempDeviationHolder &10
SET bFaultTemperatureDeviation
; rung 41
LD=(300) HMI_Current_Screen &32  ; Screen number of current screen
AND HMI_Tool_Up_Command
RSET HMI_Heat_PM  ; Heat PB on HMI

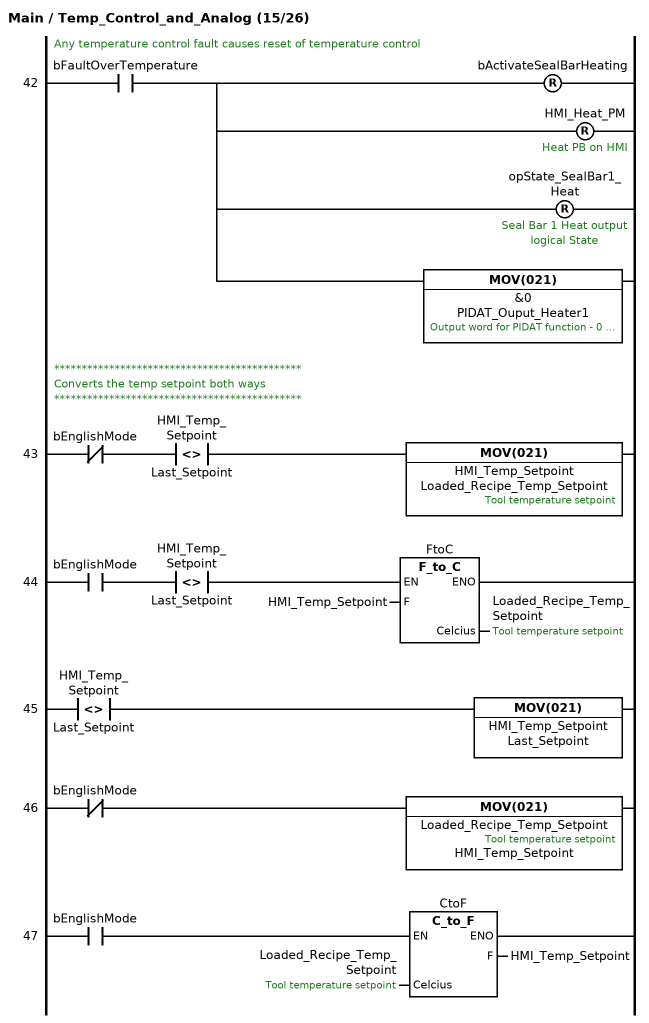
; rung 42: Any temperature control fault causes reset of temperature control
LD bFaultOverTemperature
RSET bActivateSealBarHeating
RSET HMI_Heat_PM  ; Heat PB on HMI
RSET opState_SealBar1_Heat  ; Seal Bar 1 Heat output logical State
MOV(021) &0 PIDAT_Ouput_Heater1  ; Output word for PIDAT function - 0 - 8191 range (13 bits)
; rung 43: ********************************************* / Converts the temp setpoint both ways / *********************************************
LDNOT bEnglishMode
AND<>(305) HMI_Temp_Setpoint Last_Setpoint
MOV(021) HMI_Temp_Setpoint Loaded_Recipe_Temp_Setpoint  ; Tool temperature setpoint
; rung 44
LD bEnglishMode
AND<>(305) HMI_Temp_Setpoint Last_Setpoint
CALL FtoC : F_to_C (F := HMI_Temp_Setpoint, Celcius => Loaded_Recipe_Temp_Setpoint)  ; Tool temperature setpoint
; rung 45
LD<>(305) HMI_Temp_Setpoint Last_Setpoint
MOV(021) HMI_Temp_Setpoint Last_Setpoint
; rung 46
LDNOT bEnglishMode
MOV(021) Loaded_Recipe_Temp_Setpoint HMI_Temp_Setpoint  ; Tool temperature setpoint
; rung 47
LD bEnglishMode
CALL CtoF : C_to_F (Celcius := Loaded_Recipe_Temp_Setpoint, F => HMI_Temp_Setpoint)  ; Tool temperature setpoint

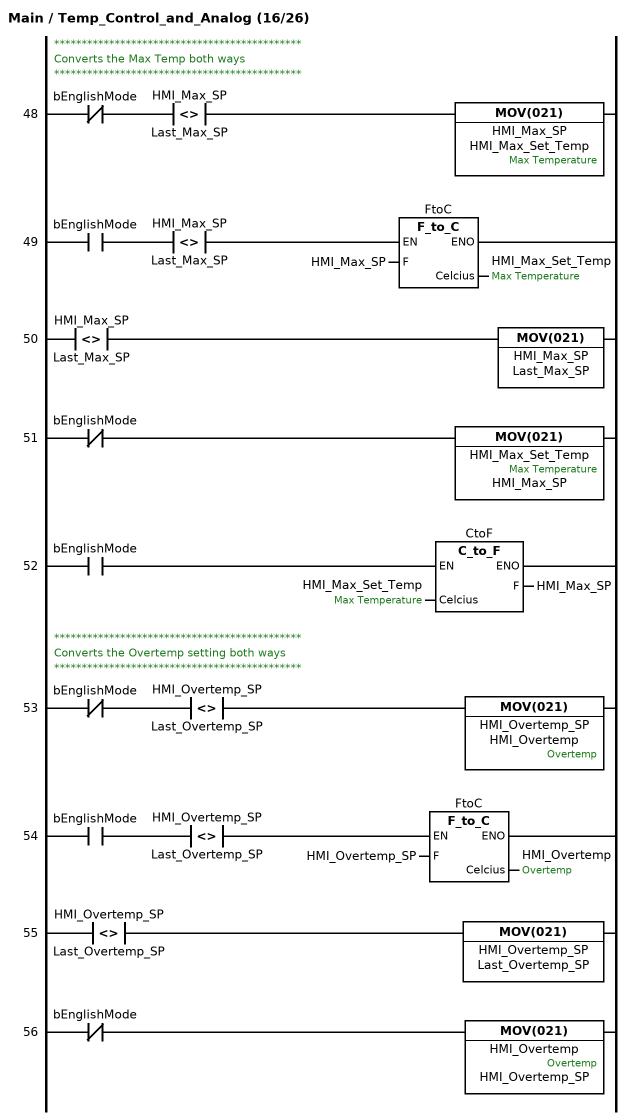
; rung 48: ********************************************* / Converts the Max Temp both ways / *********************************************
LDNOT bEnglishMode
AND<>(305) HMI_Max_SP Last_Max_SP
MOV(021) HMI_Max_SP HMI_Max_Set_Temp  ; Max Temperature
; rung 49
LD bEnglishMode
AND<>(305) HMI_Max_SP Last_Max_SP
CALL FtoC : F_to_C (F := HMI_Max_SP, Celcius => HMI_Max_Set_Temp)  ; Max Temperature
; rung 50
LD<>(305) HMI_Max_SP Last_Max_SP
MOV(021) HMI_Max_SP Last_Max_SP
; rung 51
LDNOT bEnglishMode
MOV(021) HMI_Max_Set_Temp HMI_Max_SP  ; Max Temperature
; rung 52
LD bEnglishMode
CALL CtoF : C_to_F (Celcius := HMI_Max_Set_Temp, F => HMI_Max_SP)  ; Max Temperature
; rung 53: ********************************************* / Converts the Overtemp setting both ways / *********************************************
LDNOT bEnglishMode
AND<>(305) HMI_Overtemp_SP Last_Overtemp_SP
MOV(021) HMI_Overtemp_SP HMI_Overtemp  ; Overtemp
; rung 54
LD bEnglishMode
AND<>(305) HMI_Overtemp_SP Last_Overtemp_SP
CALL FtoC : F_to_C (F := HMI_Overtemp_SP, Celcius => HMI_Overtemp)  ; Overtemp
; rung 55
LD<>(305) HMI_Overtemp_SP Last_Overtemp_SP
MOV(021) HMI_Overtemp_SP Last_Overtemp_SP
; rung 56
LDNOT bEnglishMode
MOV(021) HMI_Overtemp HMI_Overtemp_SP  ; Overtemp

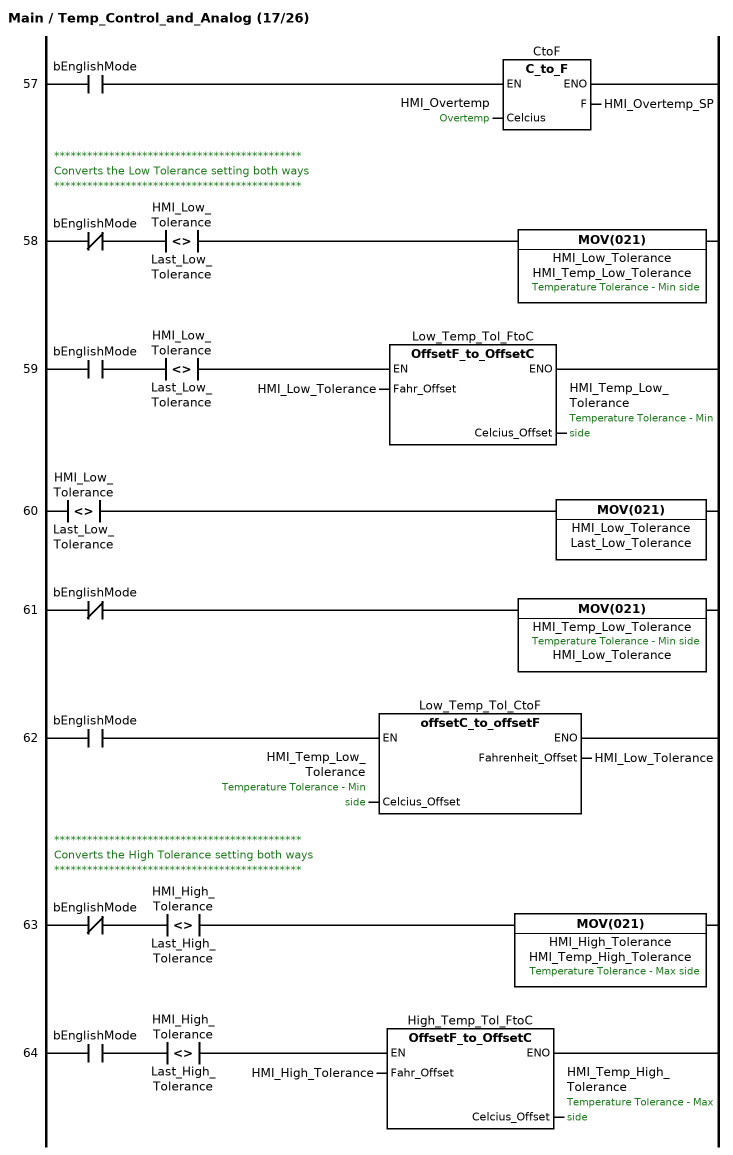
; rung 57
LD bEnglishMode
CALL CtoF : C_to_F (Celcius := HMI_Overtemp, F => HMI_Overtemp_SP)  ; Overtemp
; rung 58: ********************************************* / Converts the Low Tolerance setting both ways / *********************************************
LDNOT bEnglishMode
AND<>(305) HMI_Low_Tolerance Last_Low_Tolerance
MOV(021) HMI_Low_Tolerance HMI_Temp_Low_Tolerance  ; Temperature Tolerance - Min side
; rung 59
LD bEnglishMode
AND<>(305) HMI_Low_Tolerance Last_Low_Tolerance
CALL Low_Temp_Tol_FtoC : OffsetF_to_OffsetC (Fahr_Offset := HMI_Low_Tolerance, Celcius_Offset => HMI_Temp_Low_Tolerance)  ; Temperature Tolerance - Min side
; rung 60
LD<>(305) HMI_Low_Tolerance Last_Low_Tolerance
MOV(021) HMI_Low_Tolerance Last_Low_Tolerance
; rung 61
LDNOT bEnglishMode
MOV(021) HMI_Temp_Low_Tolerance HMI_Low_Tolerance  ; Temperature Tolerance - Min side
; rung 62
LD bEnglishMode
CALL Low_Temp_Tol_CtoF : offsetC_to_offsetF (Celcius_Offset := HMI_Temp_Low_Tolerance, Fahrenheit_Offset => HMI_Low_Tolerance)  ; Temperature Tolerance - Min side
; rung 63: ********************************************* / Converts the High Tolerance setting both ways / *********************************************
LDNOT bEnglishMode
AND<>(305) HMI_High_Tolerance Last_High_Tolerance
MOV(021) HMI_High_Tolerance HMI_Temp_High_Tolerance  ; Temperature Tolerance - Max side
; rung 64
LD bEnglishMode
AND<>(305) HMI_High_Tolerance Last_High_Tolerance
CALL High_Temp_Tol_FtoC : OffsetF_to_OffsetC (Fahr_Offset := HMI_High_Tolerance, Celcius_Offset => HMI_Temp_High_Tolerance)  ; Temperature Tolerance - Max side

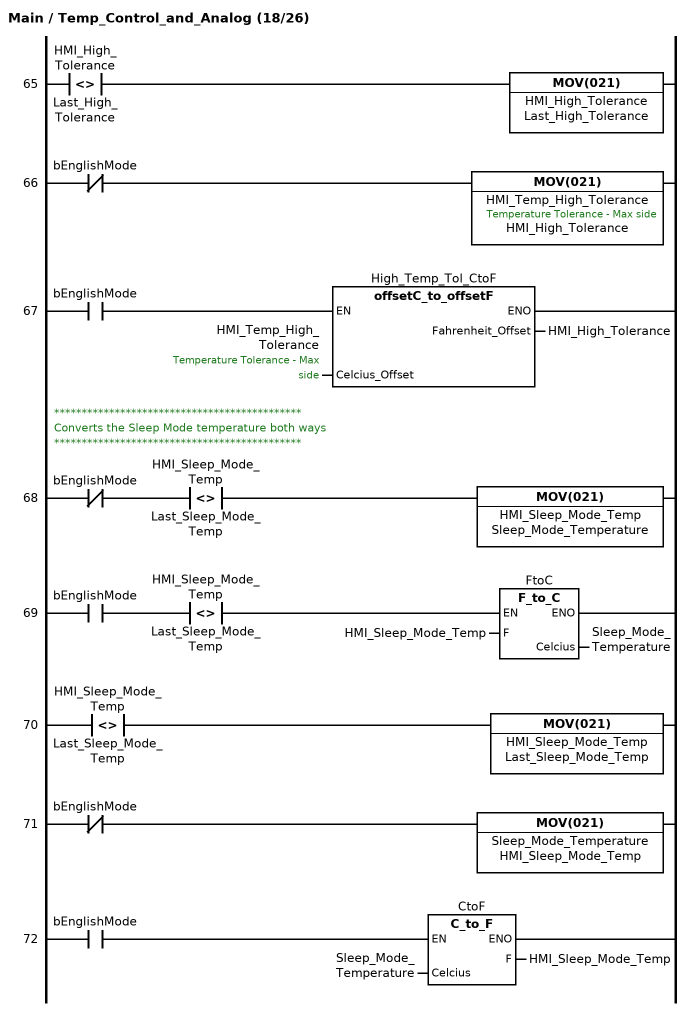
; rung 65
LD<>(305) HMI_High_Tolerance Last_High_Tolerance
MOV(021) HMI_High_Tolerance Last_High_Tolerance
; rung 66
LDNOT bEnglishMode
MOV(021) HMI_Temp_High_Tolerance HMI_High_Tolerance  ; Temperature Tolerance - Max side
; rung 67
LD bEnglishMode
CALL High_Temp_Tol_CtoF : offsetC_to_offsetF (Celcius_Offset := HMI_Temp_High_Tolerance, Fahrenheit_Offset => HMI_High_Tolerance)  ; Temperature Tolerance - Max side
; rung 68: ********************************************* / Converts the Sleep Mode temperature both ways / *********************************************
LDNOT bEnglishMode
AND<>(305) HMI_Sleep_Mode_Temp Last_Sleep_Mode_Temp
MOV(021) HMI_Sleep_Mode_Temp Sleep_Mode_Temperature
; rung 69
LD bEnglishMode
AND<>(305) HMI_Sleep_Mode_Temp Last_Sleep_Mode_Temp
CALL FtoC : F_to_C (F := HMI_Sleep_Mode_Temp, Celcius => Sleep_Mode_Temperature)
; rung 70
LD<>(305) HMI_Sleep_Mode_Temp Last_Sleep_Mode_Temp
MOV(021) HMI_Sleep_Mode_Temp Last_Sleep_Mode_Temp
; rung 71
LDNOT bEnglishMode
MOV(021) Sleep_Mode_Temperature HMI_Sleep_Mode_Temp
; rung 72
LD bEnglishMode
CALL CtoF : C_to_F (Celcius := Sleep_Mode_Temperature, F => HMI_Sleep_Mode_Temp)

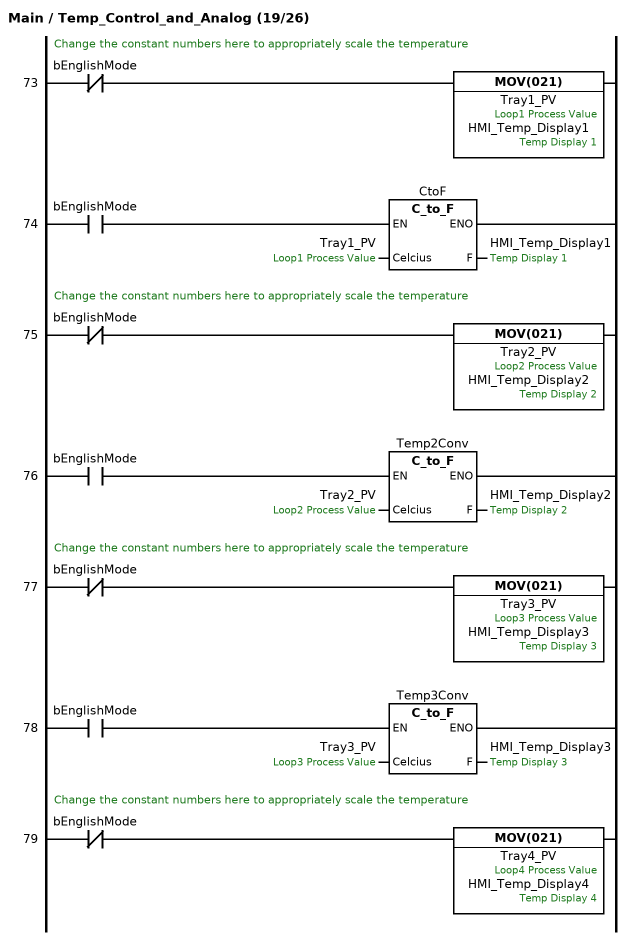
; rung 73: Change the constant numbers here to appropriately scale the temperature
LDNOT bEnglishMode
MOV(021) Tray1_PV HMI_Temp_Display1  ; Loop1 Process Value, Temp Display 1
; rung 74
LD bEnglishMode
CALL CtoF : C_to_F (Celcius := Tray1_PV, F => HMI_Temp_Display1)  ; Loop1 Process Value, Temp Display 1
; rung 75: Change the constant numbers here to appropriately scale the temperature
LDNOT bEnglishMode
MOV(021) Tray2_PV HMI_Temp_Display2  ; Loop2 Process Value, Temp Display 2
; rung 76
LD bEnglishMode
CALL Temp2Conv : C_to_F (Celcius := Tray2_PV, F => HMI_Temp_Display2)  ; Loop2 Process Value, Temp Display 2
; rung 77: Change the constant numbers here to appropriately scale the temperature
LDNOT bEnglishMode
MOV(021) Tray3_PV HMI_Temp_Display3  ; Loop3 Process Value, Temp Display 3
; rung 78
LD bEnglishMode
CALL Temp3Conv : C_to_F (Celcius := Tray3_PV, F => HMI_Temp_Display3)  ; Loop3 Process Value, Temp Display 3
; rung 79: Change the constant numbers here to appropriately scale the temperature
LDNOT bEnglishMode
MOV(021) Tray4_PV HMI_Temp_Display4  ; Loop4 Process Value, Temp Display 4

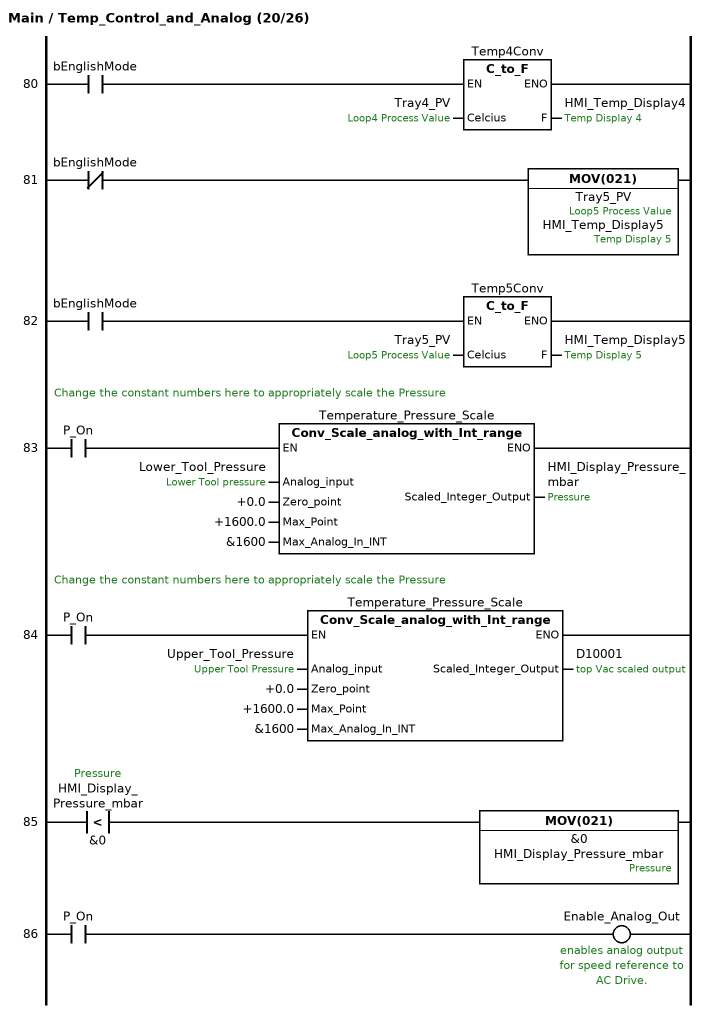
; rung 80
LD bEnglishMode
CALL Temp4Conv : C_to_F (Celcius := Tray4_PV, F => HMI_Temp_Display4)  ; Loop4 Process Value, Temp Display 4
; rung 81
LDNOT bEnglishMode
MOV(021) Tray5_PV HMI_Temp_Display5  ; Loop5 Process Value, Temp Display 5
; rung 82
LD bEnglishMode
CALL Temp5Conv : C_to_F (Celcius := Tray5_PV, F => HMI_Temp_Display5)  ; Loop5 Process Value, Temp Display 5
; rung 83: Change the constant numbers here to appropriately scale the Pressure
LD P_On
CALL Temperature_Pressure_Scale : Conv_Scale_analog_with_Int_range (Analog_input := Lower_Tool_Pressure, Zero_point := +0.0, Max_Point := +1600.0, Max_Analog_In_INT := &1600, Scaled_Integer_Output => HMI_Display_Pressure_mbar)  ; Lower Tool pressure, Pressure
; rung 84: Change the constant numbers here to appropriately scale the Pressure
LD P_On
CALL Temperature_Pressure_Scale : Conv_Scale_analog_with_Int_range (Analog_input := Upper_Tool_Pressure, Zero_point := +0.0, Max_Point := +1600.0, Max_Analog_In_INT := &1600, Scaled_Integer_Output => D10001)  ; Upper Tool Pressure, top Vac scaled output
; rung 85
LD<S(312) HMI_Display_Pressure_mbar &0  ; Pressure
MOV(021) &0 HMI_Display_Pressure_mbar  ; Pressure
; rung 86
LD P_On
OUT Enable_Analog_Out  ; enables analog output for speed reference to AC Drive.

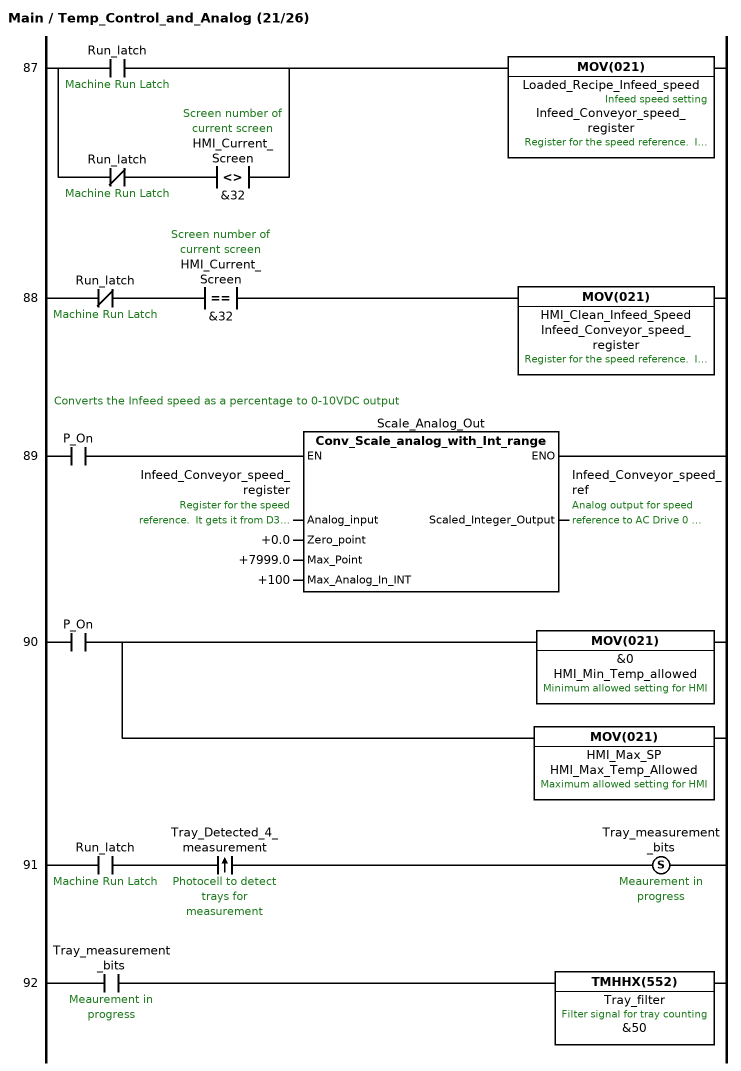
; rung 87
LD Run_latch  ; Machine Run Latch
LDNOT Run_latch  ; Machine Run Latch
AND<>(305) HMI_Current_Screen &32  ; Screen number of current screen
ORLD
MOV(021) Loaded_Recipe_Infeed_speed Infeed_Conveyor_speed_register  ; Infeed speed setting, Register for the speed reference.  It gets it from D34 or D874 for normal operation or Clean Mode
; rung 88
LDNOT Run_latch  ; Machine Run Latch
AND=(300) HMI_Current_Screen &32  ; Screen number of current screen
MOV(021) HMI_Clean_Infeed_Speed Infeed_Conveyor_speed_register  ; Register for the speed reference.  It gets it from D34 or D874 for normal operation or Clean Mode
; rung 89: Converts the Infeed speed as a percentage to 0-10VDC output
LD P_On
CALL Scale_Analog_Out : Conv_Scale_analog_with_Int_range (Analog_input := Infeed_Conveyor_speed_register, Zero_point := +0.0, Max_Point := +7999.0, Max_Analog_In_INT := +100, Scaled_Integer_Output => Infeed_Conveyor_speed_ref)  ; Register for the speed reference.  It gets it from D34 or D874 for normal operation or Clean Mode, Analog output for speed reference to AC Drive 0 - 7999 = 0 - 10VDC
; rung 90
LD P_On
MOV(021) &0 HMI_Min_Temp_allowed  ; Minimum allowed setting for HMI
MOV(021) HMI_Max_SP HMI_Max_Temp_Allowed  ; Maximum allowed setting for HMI
; rung 91
LD Run_latch  ; Machine Run Latch
@AND Tray_Detected_4_measurement  ; Photocell to detect trays for measurement
SET Tray_measurement_bits  ; Meaurement in progress
; rung 92
LD Tray_measurement_bits  ; Meaurement in progress
TMHHX(552) Tray_filter &50  ; Filter signal for tray counting

